TYPE "ADP: Decoded: Color"
VERSION : 0.1
   STRUCT
      black : String[8] := 'black';
      blue : String[8] := 'blue';
      green : String[8] := 'green';
      mix_1 : String[8] := 'mix 1';
      mix_2 : String[8] := 'mix 2';
      mix_3 : String[8] := 'mix 3';
      mix_4 : String[8] := 'mix 4';
      red : String[8] := 'red';
      white : String[8] := 'white';
      yellow : String[8] := 'yellow';
   END_STRUCT;

END_TYPE

TYPE "ADP: Encoded: Formatting: Color"
VERSION : 0.1
   STRUCT
      black { S7_SetPoint := 'True'} : String[5] := '$1C0';
      blue : String[5] := '$1C8';
      green : String[5] := '$1C2';
      mix_1 : String[5] := '$1C4';
      mix_2 : String[5] := '$1C5';
      mix_3 : String[5] := '$1C6';
      mix_4 : String[5] := '$1CY';
      red : String[5] := '$1C1';
      white : String[5] := '$1C9';
      yellow : String[5] := '$1C3';
   END_STRUCT;

END_TYPE

FUNCTION "ADP.Encode.Color" : String
{ S7_Optimized_Access := 'TRUE' }
VERSION : 0.1
   VAR_INPUT
      color : String;
      decoded : "ADP: Decoded: Color";
      encoded : "ADP: Encoded: Formatting: Color";
   END_VAR

   VAR_TEMP
      _return : String;
   END_VAR

   VAR CONSTANT
      black : String := 'BLACK';
      blue : String := 'BLUE';
      green : String := 'GREEN';
      m1 : String := 'MIX 1';
      m2 : String := 'MIX 2';
      m3 : String := 'MIX 3';
      m4 : String := 'MIX 4';
      red : String := 'RED';
      white : String := 'WHITE';
      yellow : String := 'YELLOW';
   END_VAR


BEGIN
	IF #color = #decoded.black THEN
	    #_return := #encoded.black;
	    GOTO RTRN;
	END_IF;
	IF #color = #decoded.blue THEN
	    #_return := #encoded.blue;
	    GOTO RTRN;
	END_IF;
	IF #color = #decoded.green THEN
	    #_return := #encoded.green;
	    GOTO RTRN;
	END_IF;
	IF #color = #decoded.mix_1 THEN
	    #_return := #encoded.mix_1;
	    GOTO RTRN;
	END_IF;
	IF #color = #decoded.mix_2 THEN
	    #_return := #encoded.mix_2;
	    GOTO RTRN;
	END_IF;
	IF #color = #decoded.mix_3 THEN
	    #_return := #encoded.mix_3;
	    GOTO RTRN;
	END_IF;
	IF #color = #decoded.mix_4 THEN
	    #_return := #encoded.mix_4;
	    GOTO RTRN;
	END_IF;
	IF #color = #decoded.red THEN
	    #_return := #encoded.red;
	    GOTO RTRN;
	END_IF;
	IF #color = #decoded.white THEN
	    #_return := #encoded.white;
	    GOTO RTRN;
	END_IF;
	IF #color = #decoded.yellow THEN
	    #_return := #encoded.yellow;
	    GOTO RTRN;
	END_IF;
	RTRN:
	#"ADP: Encode: Color" := #_return;
END_FUNCTION

